FUNCTION_BLOCK VfdMotor EXTENDS BasicMotor IMPLEMENTS Motor

VAR
    motorFrequency : REAL := 0.0; 
END_VAR


METHOD SetSpeed : BOOL
VAR_INPUT
	newFreq	: REAL;
END_VAR
motorFrequency := newFreq;
    SetSpeed := TRUE;
END_METHOD

END_FUNCTION_BLOCK

(* stored: Version 1.1.0.1, ProductVersion 3.1.4024.16
   POU VfdMotor: Id {e09ba69b-f0a4-4dae-a3c7-f7e65e5a9b5e}, SpecialFunc None
   Method SetSpeed: Id {55e2fb3e-843e-4aae-a188-03f4ed89549d} *)
